Staubli VAL3: kernel.pjx

--- kernel.pjx ---
Parameters version=s7.7.2 stackSize=100000 millimeterUnit=true
Program file=_control.pgx
Program file=_cycle.pgx
Program file=_interface.pgx
Program file=_interfacePoint.pgx
Program file=_kill.pgx
Program file=_plc.pgx
Program file=_pointStep.pgx
Program file=_remote.pgx
Program file=_startCycle.pgx
Program file=_startSimul.pgx
Program file=_stopCycle.pgx
Program file=_stopSimul.pgx
Program file=_taskControl.pgx
Program file=action_buffer.pgx
Program file=action_bufferT.pgx
Program file=action_do.pgx
Program file=action_resume.pgx
Program file=action_suspend.pgx
Program file=action_wait.pgx
Program file=cycle_autoON.pgx
Program file=cycle_doEvent.pgx
Program file=cycle_init.pgx
Program file=cycle_isCallUse.pgx
Program file=cycle_run.pgx
Program file=cycle_simul.pgx
Program file=cycle_start.pgx
Program file=cycle_version.pgx
Program file=cycle_waitEmpty.pgx
Program file=memory_instr.pgx
Program file=memory_loadPage.pgx
Program file=memory_onEnd.pgx
Program file=memory_onRun.pgx
Program file=memory_onStop.pgx
Program file=memory_path.pgx
Program file=memory_reLoad.pgx
Program file=memory_showAll.pgx
Program file=memory_startUp.pgx
Program file=outOfRange.pgx
Program file=remote_isHome.pgx
Program file=remote_it.pgx
Program file=remote_loadHome.pgx
Program file=remote_rstLight.pgx
Program file=start.pgx
Program file=stop.pgx
Data file=kernel.dtx
Library alias=OnEvent path=Disk://OnEvent/OnEvent.pjx autoload=true password=
Library alias=saveData path=Disk://saveData/saveData.pjx autoload=true password=
Library alias=language path=Disk://kernel/language/language.pjx autoload=true password=
Library alias=use path=Disk://kernel/userPage/userPage.pjx autoload=true password=
Library alias=plc path=Disk://PLC/PLC.pjx autoload=true password=
Library alias=cycleStatus path=Disk://cycleStatus/cycleStatus.pjx autoload=true password=
Library alias=processList path=Disk://kernel/processList/processList.pjx autoload=true password=
Library alias=interface path=Disk://kernel/template/page/page.pjx autoload=true password=
Library alias=point_interface path=Disk://trajectory/page_trajectory/page_trajectory.pjx autoload=true password=
Library alias=inOut path=Disk://saveInputOutput/saveInputOutput.pjx autoload=true password=
Library alias=prog path=Disk://instruction/PROG/PROG.pjx autoload=true password=
Library alias=page0 path=./template/page/page.pjx autoload=true password=
Library alias=page1 path=./template/page/page.pjx autoload=true password=
Library alias=page2 path=./template/page/page.pjx autoload=true password=
Library alias=page3 path=./template/page/page.pjx autoload=true password=
Library alias=page4 path=./template/page/page.pjx autoload=true password=
Library alias=page5 path=./template/page/page.pjx autoload=true password=
Library alias=page6 path=./template/page/page.pjx autoload=true password=
Library alias=page7 path=./template/page/page.pjx autoload=true password=
Library alias=page8 path=./template/page/page.pjx autoload=true password=
Library alias=page9 path=./template/page/page.pjx autoload=true password=
Library alias=page10 path=./template/page/page.pjx autoload=true password=
Library alias=page11 path=./template/page/page.pjx autoload=true password=
Library alias=page12 path=./template/page/page.pjx autoload=true password=
Library alias=page13 path=./template/page/page.pjx autoload=true password=
Library alias=page14 path=./template/page/page.pjx autoload=true password=
Library alias=page15 path=./template/page/page.pjx autoload=true password=
Library alias=page16 path=./template/page/page.pjx autoload=true password=
Library alias=page17 path=./template/page/page.pjx autoload=true password=
Library alias=page18 path=./template/page/page.pjx autoload=true password=
Library alias=page19 path=./template/page/page.pjx autoload=true password=
Library alias=page20 path=./template/page/page.pjx autoload=true password=
Library alias=page21 path=./template/page/page.pjx autoload=true password=
Library alias=page22 path=./template/page/page.pjx autoload=true password=
Library alias=page23 path=./template/page/page.pjx autoload=true password=
Library alias=page24 path=./template/page/page.pjx autoload=true password=
Library alias=page25 path=./template/page/page.pjx autoload=true password=
Library alias=instr0 path=Disk://../templates/instruction/instruction.pjx autoload=true password=
Library alias=instr19 path=Disk://../templates/instruction/instruction.pjx autoload=true password=
Library alias=instr1 path=Disk://../templates/instruction/instruction.pjx autoload=true password=
Library alias=instr2 path=Disk://../templates/instruction/instruction.pjx autoload=true password=
Library alias=instr3 path=Disk://../templates/instruction/instruction.pjx autoload=true password=
Library alias=instr4 path=Disk://../templates/instruction/instruction.pjx autoload=true password=
Library alias=instr5 path=Disk://../templates/instruction/instruction.pjx autoload=true password=
Library alias=instr6 path=Disk://../templates/instruction/instruction.pjx autoload=true password=
Library alias=instr7 path=Disk://../templates/instruction/instruction.pjx autoload=true password=
Library alias=instr8 path=Disk://../templates/instruction/instruction.pjx autoload=true password=
Library alias=instr9 path=Disk://../templates/instruction/instruction.pjx autoload=true password=
Library alias=instr10 path=Disk://../templates/instruction/instruction.pjx autoload=true password=
Library alias=instr11 path=Disk://../templates/instruction/instruction.pjx autoload=true password=
Library alias=instr12 path=Disk://../templates/instruction/instruction.pjx autoload=true password=
Library alias=instr13 path=Disk://../templates/instruction/instruction.pjx autoload=true password=
Library alias=instr14 path=Disk://../templates/instruction/instruction.pjx autoload=true password=
Library alias=instr15 path=Disk://../templates/instruction/instruction.pjx autoload=true password=
Library alias=instr16 path=Disk://../templates/instruction/instruction.pjx autoload=true password=
Library alias=instr17 path=Disk://../templates/instruction/instruction.pjx autoload=true password=
Library alias=instr18 path=Disk://../templates/instruction/instruction.pjx autoload=true password=
Library alias=page path=./template/page/page.pjx autoload=true password=
Library alias=jHome path=./template/session/saveTraj/HOME/HOME.pjx autoload=true password=
Library alias=instr20 path=Disk://../templates/instruction/instruction.pjx autoload=true password=
Library alias=instr21 path=Disk://../templates/instruction/instruction.pjx autoload=true password=
Library alias=instr22 path=Disk://../templates/instruction/instruction.pjx autoload=true password=
Library alias=instr23 path=Disk://../templates/instruction/instruction.pjx autoload=true password=
Library alias=instr24 path=Disk://../templates/instruction/instruction.pjx autoload=true password=
Library alias=instr25 path=Disk://../templates/instruction/instruction.pjx autoload=true password=
Library alias=instr26 path=Disk://../templates/instruction/instruction.pjx autoload=true password=
Library alias=instr27 path=Disk://../templates/instruction/instruction.pjx autoload=true password=
Library alias=instr28 path=Disk://../templates/instruction/instruction.pjx autoload=true password=
Library alias=instr29 path=Disk://../templates/instruction/instruction.pjx autoload=true password=
Library alias=saveInOut path=Disk://saveInputOutput/saveInputOutput.pjx autoload=true password=
Type name=ActionItem path=./template/ActionItem/ActionItem.pjx
Type name=Instruction path=./template/Instruction/Instruction.pjx
Type name=InstrItem path=Disk://kernel/template/InstrItem/InstrItem.pjx
Type name=progItem path=./template/progItem/progItem.pjx
Type name=Trajectory path=./template/Trajectory/Trajectory.pjx
Type name=dioItem path=./template/dioItem/dioItem.pjx
Type name=TrajJointItem path=./template/TrajJointItem/TrajJointItem.pjx
Type name=TrajHome path=./template/TrajHome/TrajHome.pjx

--- kernel.dtx ---
bool bEdge[5]
bool bEmergency
bool bErrorLoading
bool bHold
bool bPowered
bool bQuit
bool bRestartMove
bool bTaskPoint
bool bTimeOut
bool bWait
num nCycleStep = 4
num nLastWorkingM = 1
num nPLCClock = 7973.286
num nRemoteClock = 7973.286
num nRemoteID = -1
num nTimeOut = 10
progItem pProg
  [0]
    InstrItem iEvent
      [0]
        string sData
        string sType
    string sID
string language
string sInstr
string sItem = "JOINT @HOME"
string sMessage
string sName
string sPageLoad
string sPath
string sPathInstr
string sPathTemplate = "Disk://kernel/template/"
string sRemoteID
string sVersion[13]
  [0] = "VAL3 - s6.3.1"
  [1] = "Option testMode - demo"
  [2] = "Option valPlast - demo"
  [3] = "Configuration - D24265574A"
  [4] = "SerialNumber - ?"
  [5] = "Arm - tx90-S1-R4"
  [6] = "ArmSerialNumber - ?"
  [7] = "EP - s6.3"
  [8] = "SCA - s6.3"
  [9] = "PLC - s6.3"
  [10] = "Options - s6.3"
  [11] = "Relbo - s6.2"
  [12] = "Relbo - s5.3.2"

--- start.pgx ---
public program start()
  local num i
  local num l_nKey
  local string l_sMessage
begin
  // set the language
  call language:setLanguage(language:libPath()+"/"+saveData:language)
  // check if the robot is calibrated
  if isCalibrated()
    // FIRST BOOT
    if saveData:bInitAll
      call inOut:resetAll()
    endIf
    // INIT
    title("")
    setTextMode(0)
    userPage()
    cls()
    // SEARCH AND LOAD THE INSTRUCTION
    call language:message(l_sMessage,13)
    call use:strfill(l_sMessage,36,l_sMessage)
    call use:type(0,13,l_sMessage)
    do
      delay(0.5)
      call use:type(36+i,13,".")
      i=(i+1)
      l_nKey=getKey()
    until i==4 or l_nKey==255
    // clear the 13 line
    call use:clear(0,13)
    // look for the escape button
    if l_nKey==255 or saveData:bInitAll
      //  search for new instruction
      call language:message(l_sMessage,14)
      call use:type(2,1,l_sMessage)
      taskCreate "BuildInstr",100,memory_instr(true)
      saveData:bInitAll=false
    else
      // load in the memory the instruction
      call language:message(l_sMessage,15)
      call use:type(2,1,l_sMessage)
      taskCreate "BuildInstr",100,memory_instr(false)
    endIf
    // wait all instruction all well build
    do
      delay(0.5)
      call use:type(30+i,1,".    ")
      i=(i+1)%5
      if taskStatus("BuildInstr")>1
        taskKill("BuildInstr")
        bErrorLoading=true
        logMsg("[KERNEL] SUPERVISOR: error on loading Instruction")
        return
      endIf
    until taskStatus("BuildInstr")==-1
    // init all the variable use to comunicate with the SuperV
    cycleStatus:nToSuperV=-2
    cycleStatus:nInterfaceToSV=-2
    nRemoteID=-2
    plc:nToSuperV=-2
    // CYCLE INIT
    call cycleStatus:init()
    //
    // TASK
    //
    // CUSTOM TASK
    call OnEvent:OnStartup()
    // INTERFACE
    $jogPage(false)
    interface:libLoad("kernel/page/home")
    call use:type(1,6," Loading TASK Interface ")
    taskCreate "Interface",60,interface:main()
    wait(taskStatus("Interface")==1)
    // REMOTE
    call use:type(1,7," Loading TASK Remote ")
    taskCreate "Remote",20,remote_it()
    wait(taskStatus("Remote")==1)
    // PLC
    saveData:bPlc=true
    if saveData:bPlc==true
      call use:type(1,8," Loading TASK PLC ")
      taskCreate "Plc",50,plc:Main()
      wait(taskStatus("Plc")==1)
    endIf
    // START ALL
    cycleStatus:nToSuperV=-1
    cycleStatus:nInterfaceToSV=-1
    nRemoteID=-1
    plc:nToSuperV=-1
    //
    do
      /////////////////////////////////////////////////////
      // COMUNICATION between tha TASK
      /////////////////////////////////////////////////////
      // INTERFACE
      call _interface()
      // CYCLE
      call _cycle()
      // PLC
      if saveData:bPlc
        call _plc()
      endIf
      // REMOTE
      call _remote()
      //////////////////////
      // CONTROL
      //////////////////////
      // TASK PROBLEM
      call _taskControl()
      // CONTROL
      call _control()
      //////////////////////
      // OTHER
      //////////////////////
      // point step control
      call _pointStep()
      // CUSTOM control
      call OnEvent:control()
      // interface management
      call _interfacePoint()
      delay(0)
      //
    until bQuit
  else
    // ROBOT NOT CALIBRATED
    call language:message(l_sMessage,16)
    popUpMsg(l_sMessage)
    bErrorLoading=true
    return
  endIf
  // bye
  call _kill()
end

--- _control.pgx ---
program _control()
  local bool l_bCycle
  local bool l_bSimulation
  local num l_nID
  local num l_nResult
  local string l_sEmpty
  local string l_sMessage[2]
  local string l_sProg
begin
  //
  // load in advance to keep time
  //
  if !cycleStatus:bCycle and !cycleStatus:bSimulation and cycleStatus:bMutex==false and use:nPage>=20 and use:nPage<=29
    l_nID=0
    call processList:getCycle(l_sProg,l_nID,l_nID,0,1)
    if l_sProg!="" and !bErrorLoading
      // load the init one
      call processList:getCycle(l_sProg,l_nID,l_nID,0,0)
      if l_sProg==""
        call processList:getCycle(l_sProg,l_nID,l_nID,0,1)
      endIf
      // load it
      call prog:getProgItem(cycleStatus:pCycleProg,l_sProg)
      if cycleStatus:pCycleProg.sID==""
        // remove from the list
        bErrorLoading=true
      endIf
    elseIf l_sProg==""
      // reset the PROGRAM elements..
      resize(cycleStatus:pCycleProg.iEvent,1,1)
      cycleStatus:pCycleProg.iEvent.sType=""
      cycleStatus:pCycleProg.iEvent.sData=""
      cycleStatus:pCycleProg.sID=""
    endIf
  else
    bErrorLoading=false
  endIf
  //
  // look for the cycleStatus
  //
  if cycleStatus:bCycle
    // or cycleStatus:bSimulation
    //
    // if the working mode is not in the local or remote mode
    //
    if nLastWorkingM!=cycleStatus:nWorkingMode
      logMsg("[KERNEL] SUPERVISOR:Change working mode")
      call OnEvent:OnCycleEvent(6)
      nLastWorkingM=cycleStatus:nWorkingMode
    endIf
    // look if the power is on
    if isPowered()==false
      if bPowered
        // set the bit
        bPowered=false
        // save the last joint position if it wasn't stopped
        call cycleStatus:recordPowerDown()
        logMsg("[KERNEL] SUPERVISOR:Power off")
        call OnEvent:OnCycleEvent(7)
      endIf
    else
      bPowered=true
    endIf
    //
    // if the robot was moving and you release the hold key
    //
    if cycleStatus:nWorkingStatus==2 and cycleStatus:nPoint>0
      if !bHold
        logMsg("[KERNEL] SUPERVISOR:Release move Hold")
        call OnEvent:OnCycleEvent(0)
        bHold=true
      endIf
    else
      if cycleStatus:nWorkingStatus!=2
        bHold=false
      endIf
    endIf
    //
    // check the emergency
    //
    if esStatus()==2
      if !bEmergency
        bEmergency=true
        // look if the emergency is active
        call language:message(l_sMessage,222)
        popUpMsg(l_sMessage)
        call OnEvent:OnCycleEvent(1)
        logMsg("[KERNEL] SUPERVISOR:Emergence press")
        if saveData:bStopToPowerOff
          if cycleStatus:bCycle
            // CYCLE
            call _stopCycle()
          elseIf cycleStatus:bSimulation
            // SIMULATION
            call _stopSimul()
          endIf
          return
        endIf
      endIf
    else
      bEmergency=false
    endIf
  else
    // RESET ALL THE BIT
    bPowered=false
    bEmergency=false
    bHold=false
    nLastWorkingM=cycleStatus:nWorkingMode
    // check if already home -> reset the jPowerDown
    if cycleStatus:bIsHome
      call cycleStatus:recordPowerDown()
    endIf
  endIf
  //
  // check the restart move procedure
  //
  if !cycleStatus:bWait and !cycleStatus:bPause and !cycleStatus:bPausePLC and !cycleStatus:bStop and cycleStatus:bMoveStopped
    // restart the move
    restartMove()
    if saveData:bDebug
      ? "MOTION Restart,"+toString(".3",clock()-cycleStatus:nTime)
    endIf
    cycleStatus:bMoveStopped=false
    cycleStatus:bMotionToken=false
  else
    // stop the move
    if (cycleStatus:bWait or cycleStatus:bPause or cycleStatus:bPausePLC or cycleStatus:bStop) and !cycleStatus:bMoveStopped
      if saveData:bDebug
        ? "MOTION stopped,"+toString(".3",clock()-cycleStatus:nTime)
      endIf
      cycleStatus:bMoveStopped=true
    endIf
  endIf
  //
  // time control
  //
  // check for the resume of the task
  if bTimeOut and !cycleStatus:bPause and !cycleStatus:bPausePLC
    // resume the task
    call action_resume()
  endIf
  // is waiting
  if (cycleStatus:bWait and !cycleStatus:bPause and !cycleStatus:bPausePLC)
    if !bWait
      bTimeOut=false
      bWait=true
      nTimeOut=clock()
    endIf
    // check the time and pause the cycle
    if (clock()-nTimeOut)>saveData:nTimeOut and !bTimeOut and saveData:nTimeOut>0
      bTimeOut=true
      // suspend all the task action
      call action_suspend()
      call OnEvent:OnCycleEvent(22)
    endIf
  else
    // reset the time
    bWait=false
  endIf
  //
  // STATUS CONTROL
  //
  // save the status and the working mode of the task in global
  //
  cycleStatus:nWorkingMode=workingMode(cycleStatus:nWorkingStatus)
  cycleStatus:nEmergency=esStatus()
  // CYCLE STATUS
  l_bCycle=taskStatus("Cycle")==1 or taskStatus("Cycle")==0
  // SIMULATION STATUS
  l_bSimulation=taskStatus("Simulation")==1 or taskStatus("Simulation")==0
  //
  // REFRESH and CYCLE status
  //
  if cycleStatus:bSimulation!=l_bSimulation
    // simulation
    cycleStatus:bSimulation=l_bSimulation
    // INIT ALL
    if !l_bSimulation
      // init all
      call cycle_init()
      l_sEmpty=""
      call memory_onStop(l_sEmpty)
    endIf
    use:bUseRefresh=true
  endIf
  if cycleStatus:bCycle!=l_bCycle
    // cycle
    cycleStatus:bCycle=l_bCycle
    if !l_bCycle
      // init all
      call cycle_init()
      l_sEmpty=""
      call memory_onStop(l_sEmpty)
      // check if reload the last process List saved
      if saveData:bReloadList
        call processList:loadProcessList(l_nResult)
        if l_nResult!=0
          // message
          call language:message(l_sMessage,-7)
          call language:message(l_sMessage[1],70)
          popUpMsg(l_sMessage+" "+l_sMessage[1])
        endIf
      endIf
    endIf
    use:bUseRefresh=true
  endIf
  // check if is need to reload ALL
  if saveData:bToReload and !cycleStatus:bCycle and !cycleStatus:bSimulation
    call memory_reLoad()
    saveData:bToReload=false
  endIf
end

--- _cycle.pgx ---
program _cycle()
  local bool bActive
  local bool l_bContinue
  local bool l_bTollerance
  local string l_sMessage
begin
  bActive=false
  //
  // STOP CYCLE
  //
  if cycleStatus:bToStop
    stopMove()
    if cycleStatus:bCycle
      call _stopCycle()
    else
      // SIMULATION
      if cycleStatus:bSimulation
        call _stopSimul()
      endIf
    endIf
    //  RESET
    cycleStatus:bToStop=false
    cycleStatus:nToSuperV=-1
    //
    // HOMING
    //
  elseIf cycleStatus:bToHome
    cycleStatus:bToHome=false
    if watch(cycleStatus:bSimulation==false and cycleStatus:bCycle==false,3)
      cycleStatus:sTraj=""
      cycleStatus:iToSuperV.sType="HOME"
      cycleStatus:iToSuperV.sData="simul"
      call _startSimul(cycleStatus:iToSuperV)
    endIf
    //
    // END CYCLE
    //
  elseIf cycleStatus:bToEnd==true
    cycleStatus:bToEnd=false
    // end the cycle
    if cycleStatus:bCycle and !cycleStatus:bEnding and esStatus()!=2
      logMsg("[KERNEL] CYCLE:Ending Cycle")
      cycleStatus:bEnding=true
      call OnEvent:OnCycleEvent(4)
    endIf
    //
    // START CYCLE
    //
  elseIf cycleStatus:bToStart==true
    cycleStatus:bToStart=false
    if taskStatus("Cycle")==-1
      call _startCycle()
      logMsg("[KERNEL] SUPERVISOR:Cycle>Start cycle")
    endIf
    //
    // PAUSE / RESUME
    //
  elseIf cycleStatus:bToPause
    cycleStatus:bToPause=false
    // PAUSE
    if !cycleStatus:bPause
      // pause the robot
      cycleStatus:bPause=true
      // stop the motion
      stopMove()
      if isPowered()
        call cycleStatus:recordPowerDown()
      endIf
      logMsg("[KERNEL] CYCLE:Pause the cycle")
      // onEvent
      call OnEvent:OnCycleEvent(2)
      // resume the cycle after a pause
    elseIf cycleStatus:bPause==true and cycleStatus:bMoveStopped==true and esStatus()!=2
      // check the tollerance if not do nothing
      call cycleStatus:checkTollerance(l_bTollerance)
      if (!isPowered() and !l_bTollerance and (cycleStatus:nWorkingMode==4 or cycleStatus:nWorkingMode==3))
        logMsg("[KERNEL] CYCLE:Error on Tollerance check during RESTART")
      else
        logMsg("[KERNEL] CYCLE:Restart the cycle")
        // on Event
        call OnEvent:OnCycleEvent(3)
        // restart, reset the bit for the pause
        cycleStatus:bPause=false
      endIf
    endIf
  else
    // check the auto_ON
    if cycleStatus:bAutoON
      cycleStatus:bAutoON=false
      call cycle_autoON(l_bContinue)
    endIf
    // SWITCH
    switch cycleStatus:nToSuperV
      case 0
        //
      break
      case 1
        //
      break
      case 2
        //
      break
      case 3
        //
      break
      case 4
        // OUT OF TIME
        call language:message(l_sMessage,230)
        popUpMsg(l_sMessage)
        if cycleStatus:bCycle
          //STOP CYCLE
          call _stopCycle()
        else
          if cycleStatus:bSimulation
            // STOP SIMULATION
            call _stopSimul()
          endIf
        endIf
        bActive=true
      break
      case 6
        // PAUSE CYCLE
        call OnEvent:pauseCycle()
        bActive=true
      break
      case 7
        // RESUME CYCLE
        call OnEvent:resumeCycle()
        bActive=true
      break
      default
      break
    endSwitch
  endIf
  // release
  if bActive
    cycleStatus:nToSuperV=-1
  endIf
  //
end

--- _interface.pgx ---
program _interface()
  local bool bActive
  local bool bStop
  local num i
  local string message
  local string sString
begin
  bActive=false
  switch cycleStatus:nInterfaceToSV
    case 0
      //
      // go to the production page
      //
      logMsg("[KERNEL] SUPERVISOR:Interface>Call Production page")
      bActive=true
    break
    case 1
      //
      //  Exit from KERNEL
      //
      bQuit=true
      bActive=true
    break
    case 2
      //
      //  Simulation of a program
      //
      call _startSimul(cycleStatus:iToSuperV)
      bActive=true
    break
    case 3
      //
      //  Simulation of an Event
      //
      call _startSimul(cycleStatus:iToSuperV)
      bActive=true
    break
    case 4
      //
      //  Timer simulation
      //
      cycleStatus:iToSuperV.sType="TIMER"
      cycleStatus:iToSuperV.sData="executing"
      call _startSimul(cycleStatus:iToSuperV)
      bActive=true
    break
    //
    // PLC
    //
    case 10
      // PLC activation
      logMsg("[KERNEL] SUPERVISOR:Interface>Start the Task PLC")
      plc:nToSuperV=-2
      taskCreate "Plc",50,plc:Main()
      saveData:bPlc=true
      plc:nToSuperV=-1
      bActive=true
    break
    case 11
      // PLC de-activation
      logMsg("[KERNEL] SUPERVISOR:Interface>Kill the Task PLC")
      taskKill("Plc")
      call plc:kill()
      saveData:bPlc=false
      bActive=true
    break
    default
      //
    break
  endSwitch
  // reset
  if bActive
    cycleStatus:nInterfaceToSV=-1
  endIf
end

--- _interfacePoint.pgx ---
program _interfacePoint()
  local string l_sMessage
begin
  //
  // acces to the point interface
  //
  if isKeyPressed(289) and (taskStatus("Point")==-1 or taskStatus("Point")>1)
    if (use:nPage>=100000 and use:nPage<=100009) or (use:nPage>=10000 and use:nPage<=10009)
      // TODO
      l_sMessage="Please exit from the page editor before enter in page POINT...."
      popUpMsg(l_sMessage)
      delay(3)
    else
      // SUSPEND THE TASK INTERFACE
      taskKill("Point")
      taskSuspend("Interface")
      // POINT INTERFACE
      taskCreate "Point",50,point_interface:main()
      bTaskPoint=true
      use:bUseRefresh=true
    endIf
  elseIf (taskStatus("Interface")==0 and taskStatus("Point")==-1) and bTaskPoint
    // TASK RESUME
    bTaskPoint=false
    taskResume("Interface",0)
    use:bUseRefresh=true
  endIf
  // release
  delay(0)
end

--- _kill.pgx ---
public program _kill()
  local string l_sMessage
begin
  // KILL KERNEL
  $jogPage(true)
  title("")
  cls()
  call language:message(l_sMessage,17)
  call use:timerDialog(l_sMessage,0)
  logMsg("[KERNEL] SUPERVISOR:Interface>Quit KERNEL")
  taskKill("Interface")
  taskKill("Point")
  taskKill("Remote")
  taskKill("Cycle")
  taskKill("Plc")
  taskKill("Action")
  watch(taskStatus("Interface")==-1,1)
  watch(taskStatus("Remote")==-1,1)
  watch(taskStatus("Cycle")==-1,1)
  watch(taskStatus("Plc")==-1,1)
  // save the last setting
  saveData:libSave()
  // save the cycle
  call processList:save()
  bQuit=false
  // give a time delay
  delay(1)
end

--- _plc.pgx ---
program _plc()
  local bool bActive
begin
  // PLC
  bActive=false
  switch plc:nToSuperV
    case 0
      //
      // Start Cycle
      //
      if taskStatus("Cycle")==-1
        cycleStatus:bToStart=true
      endIf
      bActive=true
    break
  endSwitch
  //
  if bActive
    plc:nToSuperV=-1
  endIf
end

--- _pointStep.pgx ---
program _pointStep()
  local ActionItem l_aPointData
  local num l_nId
  local num l_nIdPoint
  local num l_nLastId
  local Trajectory l_tTraj
begin
  //
  //  SYNCRO the point STEP of the trajectory
  //
  //  only if on Cycle
  if (cycleStatus:bCycle or cycleStatus:bSimulation)
    // get the actual Point ID..
    call cycleStatus:getTraj(l_tTraj)
    if l_tTraj.sID!="null" and l_tTraj.sID!=""
      // check it..
      if cycleStatus:nPoint>size(l_tTraj.tSuper)-1
        // init all
        cycleStatus:nPoint=0
        call cycleStatus:removeTraj()
        //? "[POINTSTEP]: trajectory removed:"+l_tTraj.sID
      elseIf getMoveId()>l_tTraj.tSuper[cycleStatus:nPoint].nMoveId+1
        //? "[POINTSTEP]: trajectory update: "+l_tTraj.sID+toString("4",cycleStatus:nPoint)
        // put one MORE
        cycleStatus:nPoint=cycleStatus:nPoint+1
      endIf
      if !isEmpty()
        // set a traj is doing
        cycleStatus:bTraj=true
        if cycleStatus:nEvent!=l_tTraj[0].nId
          // update the EVENT ID
          cycleStatus:nEvent=l_tTraj[0].nId
          //? "[POINTSTEP]: trajectory event update: "+l_tTraj.sID+toString("4",cycleStatus:nEvent)
        endIf
        l_nId=roundDown(getMoveId())
        // refresh the percentage point distance
        cycleStatus:nIdPercentage=abs(getMoveId()-l_nId)*100
      endIf
    elseIf cycleStatus:nPoint!=0 or cycleStatus:bTraj
      // reset
      //? "[POINTSTEP]: reset the traj parameter"
      cycleStatus:bTraj=false
      cycleStatus:nPoint=0
    endIf
  else
    // reset the TRAJ
    cycleStatus:nPoint=0
    cycleStatus:bTraj=false
  endIf
  //
end

--- _remote.pgx ---
program _remote()
  local bool bActive
  local InstrItem l_iProg
  local string message
  local string sString
begin
  bActive=false
  switch nRemoteID
    case 0
      // START
      if taskStatus("Cycle")==-1
        logMsg("[KERNEL] SUPERVISOR:REMOTE>Start cycle")
        cycleStatus:bToStart=true
      endIf
      bActive=true
    break
    case 1
      //STOP
      cycleStatus:bToStop=true
      bActive=true
    break
    case 2
      //END CYCLE
      if taskStatus("Cycle")!=-1
        logMsg("[KERNEL] SUPERVISOR:REMOTE>End cycle")
        cycleStatus:bToEnd=true
      endIf
      bActive=true
    break
    case 3
      // HOME STRATEGY
      if taskStatus("Cycle")==-1
        logMsg("[KERNEL] SUPERVISOR:REMOTE>Home strategy")
        cycleStatus:bToHome=true
      endIf
      bActive=true
    break
    case 4
      // simulation of the program
      l_iProg.sType="PROG"
      l_iProg.sData=sRemoteID
      call _startSimul(l_iProg)
      logMsg("[KERNEL] SUPERVISOR:REMOTE>insert the program: "+sRemoteID)
      bActive=true
    break
  endSwitch
  if bActive
    nRemoteID=-1
    sRemoteID=""
    if taskStatus("Interface")==0
      taskResume("Interface",0)
    endIf
  endIf
end

--- _startCycle.pgx ---
program _startCycle()
  local bool l_bContinue
  local num l_nID
  local string l_sMessage
  local string l_sProcessList
begin
  // check home
  if cycleStatus:bIsHome or saveData:bNoUseHome
    // look if there are program into the process list
    if !cycleStatus:bCycle and !cycleStatus:bSimulation and esStatus()!=2
      call processList:getLoaded(l_sProcessList)
      if l_sProcessList!=""
        l_nID=0
        call processList:getCycle(l_sMessage,l_nID,l_nID,0,1)
        if l_sMessage!=""
          // Create the Cycle Task
          if taskStatus("Cycle")==-1
            // init all
            call cycleStatus:init()
            // onEvent
            cycleStatus:bCycle=true
            call OnEvent:OnCycleEvent(13)
            if cycleStatus:bToStop
              cycleStatus:bCycle=false
              return
            endIf
            // put the power ON on remote
            call cycle_autoON(l_bContinue)
            if l_bContinue
              taskCreate "Cycle",80,cycle_start()
              // start the action Task for the traj
              if taskStatus("Action")==-1
                taskCreate "Action",80,action_buffer()
              endIf
            else
              // error while starting
              cycleStatus:bCycle=false
              return
            endIf
          endIf
        else
          // ERROR no program into the process list
          call OnEvent:OnCycleEvent(9)
        endIf
      else
        // NO processList loaded
        call OnEvent:OnCycleEvent(9)
      endIf
    endIf
  else
    // the robot is not at home
    call language:message(l_sMessage,223)
    popUpMsg(l_sMessage)
  endIf
end

--- _startSimul.pgx ---
program _startSimul(InstrItem& x_iInstr (dimensions=1))
  local bool l_bContinue
  local string l_sEvent
begin
  // init all
  call cycleStatus:init()
  // CHECK FOR CYCLE EVENT
  if !cycleStatus:bCycle and !cycleStatus:bSimulation
    // set the Simulation is ON
    cycleStatus:bSimulation=true
    if x_iInstr.sType=="HOME"
      cycleStatus:bHoming=true
    endIf
    // SIMULATION
    logMsg("[KERNEL] SUPERVISOR:Interface>Simulation of the event: "+x_iInstr.sType+" "+x_iInstr.sData)
    taskCreate "Simulation",50,cycle_simul(x_iInstr)
    // start the action Task for the traj
    taskCreate "Action",80,action_buffer()
  endIf
end

--- _stopCycle.pgx ---
program _stopCycle()
  local string l_sEmpty
  local num nCycleDone
  local num nCycleToDo
  local string sProgName
begin
  // reset the bit
  // Stop the robot
  stopMove()
  if saveData:bStopToPowerOff
    disablePower()
  endIf
  logMsg("[KERNEL] SUPERVISOR:Cycle>Stop cycle")
  // kill the Task...
  taskKill("Cycle")
  taskKill("Action")
  watch(taskStatus("Cycle")==-1 and taskStatus("Action")==-1,1)
  //
  resetMotion()
  call OnEvent:OnCycleEvent(5)
  // delete the last program
  call processList:getCycle(sProgName,nCycleToDo,nCycleDone,0,1)
  if (nCycleToDo-nCycleDone)<=1
    call processList:loopMode()
  else
    call processList:setCycle(sProgName,nCycleToDo,nCycleDone+1,0,1)
  endIf
end

--- _stopSimul.pgx ---
program _stopSimul()
  local string l_sEmpty
begin
  // reset the bit
  stopMove()
  // STOP SIMULATION
  logMsg("[KERNEL] SUPERVISOR:Cycle>Stop Simulation")
  // kill the task...
  taskKill("Simulation")
  taskKill("Action")
  watch(taskStatus("Simulation")==-1 and taskStatus("Action")==-1,1)
  //
  resetMotion()
  call OnEvent:OnCycleEvent(10)
end

--- _taskControl.pgx ---
program _taskControl()
  local bool l_bRestart[2]
  local bool l_bYes
  local string l_sButton[2]
  local string l_sMessage[2]
begin
  //
  // Check the task Cycle
  //
  if taskStatus("Cycle")>1 or (cycleStatus:bCycle and taskStatus("Action")>1)
    if taskStatus("Cycle")>=150 and taskStatus("Cycle")<=154
      call outOfRange()
    else
      logMsg("[KERNEL] SUPERVISOR:Task Cycle problem")
      call OnEvent:OnCycleEvent(12)
    endIf
    call _stopCycle()
  endIf
  //
  // Check the task Simulation
  //
  if taskStatus("Simulation")>1 or (cycleStatus:bSimulation and taskStatus("Action")>1)
    if taskStatus("Simulation")>=150 and taskStatus("Simulation")<=154
      call outOfRange()
    else
      logMsg("[KERNEL] SUPERVISOR:Task Simulation problem")
      call OnEvent:OnCycleEvent(12)
    endIf
    call _stopSimul()
  endIf
  // Check the task PLC every 5 second
  if taskStatus("Plc")>1
    if clock()-nPLCClock>5
      nPLCClock=clock()
      taskResume("Plc",0)
    endIf
  else
    nPLCClock=clock()
  endIf
  // check the task remote every 5 seconds
  if taskStatus("Remote")>1
    if clock()-nRemoteClock>5
      nRemoteClock=clock()
      taskKill("Remote")
      taskCreate "Remote",20,remote_it()
    endIf
  else
    nRemoteClock=clock()
  endIf
  //
  // TASK INTERFACE
  //
  //
  // look if there is something wrong for the interface
  //
  l_bRestart=false
  if taskStatus("Interface")==61
    logMsg("[KERNEL] SUPERVISOR:WakeUpInterface> error61")
    get()
    taskResume("Interface",0)
    watch(taskStatus("Interface")==1,1)
  endIf
  //
  // look if the interface has been stopped
  //
  if cycleStatus:nInterfaceToSV==-1 and taskStatus("Simulation")==-1
    // look for the mode
    if taskStatus("Interface")>1
      call language:message(l_sMessage,221)
      call use:timerDialog(l_sMessage,1)
      // get a Key
      get()
      // RESTART ...
      logMsg("[KERNEL] SUPERVISOR:WakeUpInterface>Restart")
      call language:message(l_sMessage,220)
      call use:timerDialog(l_sMessage,1)
      taskKill("Interface")
      taskCreate "Interface",60,interface:main()
      wait(taskStatus("Interface")==1)
    endIf
  endIf
  //
  // look if the interface has been stopped
  //
  if cycleStatus:nInterfaceToSV==-1 and taskStatus("Simulation")==-1
    if taskStatus("Point")>1
      call language:message(l_sMessage,221)
      call use:timerDialog(l_sMessage,1)
      // get a Key
      get()
      // RESTART
      logMsg("[KERNEL] SUPERVISOR:WakeUpInterface>Restart Point")
      call language:message(l_sMessage,220)
      call use:timerDialog(l_sMessage,1)
      taskKill("Point")
      taskCreate "Point",50,point_interface:main()
      wait(taskStatus("Point")==1)
    endIf
  endIf
end

--- action_buffer.pgx ---
program action_buffer()
  local ActionItem l_aAction
  local bool l_bEmpty
begin
  // wait the Task Cycle or simulation has been started
  wait(cycleStatus:bCycle or cycleStatus:bSimulation)
  //
  // scan the action
  //
  while (cycleStatus:bCycle or cycleStatus:bSimulation)
    // wait to move to run STATE
    do
      // scan the action item
      call cycleStatus:isActionEmpty(l_bEmpty)
      cycleStatus:bActionRunning=!l_bEmpty
      if !(cycleStatus:bCycle or cycleStatus:bSimulation)
        return
      endIf
      delay(0)
    until l_bEmpty==false
    // execute
    call cycleStatus:getAction(l_aAction)
    call action_do(l_aAction,-1)
    // remove
    call cycleStatus:removeAction()
  endWhile
  //
end

--- action_bufferT.pgx ---
program action_bufferT(ActionItem& x_aAction[] (dimensions=1))
  local num i
  local bool l_bMutex
  local bool l_bTraj
  local num l_nActualStep
  local num l_nIdTask
  local num l_nInstrId
  local num l_nMinus
  local num l_nTask
  local num l_nZero
  local string l_sAction
  local string l_sEmpty
  local string l_sInstrType
begin
  //
  // INIT
  //
  // wait the Task Cycle or simulation has been started
  wait(cycleStatus:bCycle or cycleStatus:bSimulation)
  //
  if x_aAction.iInstr.sType!="" and x_aAction.iInstr.sType!="null"
    // compose the instruction
    // do the action
    x_aAction.nDistance=0
    x_aAction.nMoveId=-1
    x_aAction.nPointId=-1
    call action_do(x_aAction,-1)
  endIf
end

--- action_do.pgx ---
program action_do(ActionItem& x_aAction[] (dimensions=1), num x_nIndex (dimensions=1))
  local num i
  local num j
  local bool l_bExit
  local num l_nClock
  local num l_nDistance
  local num l_nResult
  local string l_sData
  local string l_sEmpty
  local string l_sInstr
  local string l_sInstruction
  local string l_sType
begin
  // check if not empty...
  if x_aAction.iInstr[0].sType!="" or x_aAction.iInstr[1].sType!="" or x_aAction.iInstr[2].sType!=""
    if saveData:bDebug
      ? "ACTION INSERT,"+x_aAction.iInstr.sType+" "+x_aAction.iInstr.sData+",ID="+toString(".3",getMoveId())+","+toString(".3",clock()-cycleStatus:nTime)+",x_ID="+toString("",x_aAction.nMoveId)+",x_Dist="+toString(".2",x_aAction.nDistance)
    endIf
    l_nClock=clock()
    // wait the correct moveID
    wait((x_aAction.nMoveId+x_aAction.nDistance)<=getMoveId() or (isEmpty()) and !cycleStatus:bPause)
    // look if there are several sAction in the traj
    for i=0 to (size(x_aAction.iInstr)-1)
      // check for not empty space
      if x_aAction.iInstr[i].sType!=""
        // get the instruction
        l_sData=x_aAction.iInstr[i].sData
        l_sType=x_aAction.iInstr[i].sType
        call saveInOut:replaceIO(l_sData,l_sType,l_sData)
        l_sInstr=l_sType+" "+l_sData
        if saveData:bDebug
          ? "ACTION RUNNING,"+l_sInstr+",ID="+toString(".3",getMoveId())+","+toString(".3",clock()-cycleStatus:nTime)+",MoveID="+toString("",x_aAction.nMoveId)+",Dist="+toString(".2",x_aAction.nDistance)
        endIf
        // PRINT LOG
        if cycleStatus:bCycle
          if x_aAction.nPointId!=-1
            // is inside a trajectory
            call cycleStatus:printLog(" ."+l_sInstr)
          else
            // is outside a trajectory
            call cycleStatus:printLog("-"+l_sInstr)
          endIf
        endIf
        cycleStatus:sToShow=l_sInstr
        cycleStatus:sLastAction=l_sInstr
        if x_aAction.nPointId==-1
          // refresh the LINE of the program...
          cycleStatus:bTraj=false
          cycleStatus:nEvent=x_nIndex
        endIf
        //
        // RUN THE ACTION
        //
        call memory_onRun(x_aAction.iInstr[i])
      endIf
    endFor
    // release
    cycleStatus:sToShow=""
  endIf
end

--- action_resume.pgx ---
program action_resume()
begin
  //
  // suspend all the task action
  //
  // check first...
  if taskStatus("Cycle")!=-1
    taskResume("Cycle",0)
  endIf
  if taskStatus("Action")!=-1
    taskResume("Action",0)
  endIf
  //..
end

--- action_suspend.pgx ---
program action_suspend()
begin
  // suspend all the task action
  if taskStatus("Cycle")!=-1
    taskSuspend("Cycle")
  endIf
  if taskStatus("Action")!=-1
    taskSuspend("Action")
  endIf
  //..

end

--- action_wait.pgx ---
program action_wait()
  local bool l_bEmpty
begin
  // wait no action on the list
  while l_bEmpty==false
    call cycleStatus:isActionEmpty(l_bEmpty)
    delay(0)
  endWhile
end

--- cycle_autoON.pgx ---
program cycle_autoON(bool& x_bResult[] (dimensions=1))
  local num i
  local bool l_bTollerance
  local num l_nClock
  local string l_sMessage
begin
  //
  // look first if is in remote mode then
  // look if it is in mode automatic and the power is ON
  //
  x_bResult=false
  //
  //  CHECK FOR STATUS MODE
  //
  // look for the remote status NB check jPowerDown
  if workingMode()==4
    // check tollerance
    call cycleStatus:checkTollerance(l_bTollerance)
    if (!isPowered() and !l_bTollerance and cycleStatus:bPause)
      logMsg("[KERNEL] CYCLE:Error on Tollerance check during AUTO ON")
    elseIf isPowered()==false and esStatus()!=2 and cycleStatus:nWorkingMode!=2
      // enable auto connect move
      autoConnectMove(true)
      // VAL3 ?? unknow
      x_bResult=true
      // power it
      enablePower()
      delay(1)
      watch((isPowered()==true or esStatus()==2),3)
      if esStatus()==2
        return
      endIf
    endIf
  elseIf workingMode()!=3
    // put the robot in AUTO MODE
    call language:message(l_sMessage,200)
    // look fot the auto mode
    call use:timerDialog(l_sMessage,2)
  elseIf workingMode()==3 and !isPowered()
    // pu the power ON
    call language:message(l_sMessage,201)
    l_nClock=clock()
    do
      call use:timerDialog(l_sMessage,0.5)
    until (clock()-l_nClock)>5 or getKey()==255 or esStatus()==2
    if isPowered()==false
      return
    endIf
  endIf
  // it's ok give it back
  if esStatus()!=2 and ((workingMode()==3 or workingMode()==4) and isPowered())
    x_bResult=true
  endIf
  //
end

--- cycle_doEvent.pgx ---
program cycle_doEvent(InstrItem x_iInstr (dimensions=1), num x_nIndex (dimensions=1))
  local ActionItem l_aAction
  local bool l_bTraj
  local num l_nId
  local num l_nOffset
  local num l_nResult
  local string l_sInstruction
  local string l_sName
  local string l_sPath
begin
  //
  // DIVIDE INTO trajectory or NOT
  //
  call saveData:getPathInstr(x_iInstr.sType,l_sPath)
  if l_sPath!=""
    // DIVIDE INSTRUCTION FROM TRAJECTORY
    if find(l_sPath,"trajectory")==-1
      // EXECUTE THE ACTION
      call action_wait()
      // UPDATE THE ACTION TO DO...
      l_aAction.nDistance=1-saveData:nRound/100
      call cycleStatus:getLastId(l_aAction.nMoveId)
      l_aAction.iInstr=x_iInstr
      l_aAction.nPointId=-1
      call action_do(l_aAction,x_nIndex)
    else
      // TRAJ
      // print the action log
      l_sInstruction=x_iInstr.sType+" "+x_iInstr.sData
      if cycleStatus:bCycle
        // set the clock end
        call cycleStatus:printLog("-"+l_sInstruction)
      endIf
      // update the LINE ID
      cycleStatus:nLastIdPoint=x_nIndex
      // run it
      call memory_onRun(x_iInstr)
    endIf
  else
    // PATH NOT FOUND
    cycleStatus:bToStop=true
  endIf
end

--- cycle_init.pgx ---
program cycle_init()
// initialization of the cycle
  local num hours
  local num i
  local num index
  local num l_nSize
begin
  //
  // watch all the instructin has been launched
  //
  // init all the mutex
  cycleStatus:bMutex=false
  // reset
  if saveData:bDebug
    logMsg("[DEBUG] CYCLE: INIT Started")
    ? "CYCLE: INIT Started "
  endIf
  //
  // init all the cyclestatus variable
  //
  call cycleStatus:init()
  //
  // reset the cycle DONE
  //
  call processList:init()
  // check the version status
  call cycle_version()
  if saveData:bDebug
    logMsg("[DEBUG] CYCLE: INIT Terminated")
    ? "CYCLE: INIT Terminated"
  endIf
  // reset all the internal BIT
  bWait=false
  bTimeOut=false
end

--- cycle_isCallUse.pgx ---
program cycle_isCallUse()
  local num l_nResult
  local progItem l_pProg
begin
  // JUMP CALL USED
  if cycleStatus:bCALL
    do
      // reset the BIT
      cycleStatus:bCALL=false
      if cycleStatus:iToSuperV.sType=="PROG"
        // load the SUB PROG
        call prog:getProgItem(pProg,cycleStatus:iToSuperV.sData)
        // check it
        if pProg.sID!=""
          call cycle_run(pProg)
        else
          // STOP ALL
          cycleStatus:bToStop=true
        endIf
        // came back and restore
      else
        // just the LINE
        call cycle_doEvent(cycleStatus:iToSuperV,0)
      endIf
      // NESTED....
    until cycleStatus:bCALL==false
  endIf
end

--- cycle_run.pgx ---
program cycle_run(progItem& x_pProgram[] (dimensions=1))
  local num i
  local num j
  local num l_nClock
  local num l_nResult
  local num l_nSize
  local progItem l_pProg
  local string l_sEvent
begin
  //
  // START
  //
  cycleStatus:nEvent=0
  cycleStatus:nPoint=0
  // refresh
  cycleStatus:pCycleProg=l_pProg=x_pProgram
  // check the cycle
  if cycleStatus:bCycle
    // print the actual program
    call cycleStatus:printLog("[PROG "+l_pProg.sID+"]")
  endIf
  l_nSize=size(l_pProg.iEvent)
  for i=0 to l_nSize-1
    // wait pause false before doing the next instruction
    wait(cycleStatus:bPause==false and isPowered() and cycleStatus:nWorkingStatus==0)
    if l_pProg.iEvent[i].sType!=""
      l_sEvent=l_pProg.iEvent[i].sType+" "+l_pProg.iEvent[i].sData
      if saveData:bDebug
        ? "ACTION READ,"+l_sEvent+",ID="+toString(".3",getMoveId())+","+toString(".3",clock()-cycleStatus:nTime)
      endIf
      call cycle_doEvent(l_pProg.iEvent[i],i)
      // JUMP CALL USED
      call cycle_isCallUse()
      // GOTO USED
      if cycleStatus:bGOTO
        // terminate this and run the GOTO
        i=l_nSize-1
      endIf
    endIf
  endFor
  // GOTO ...
  if cycleStatus:bGOTO
    // INIT
    cycleStatus:bGOTO=false
    call action_wait()
    if cycleStatus:iToSuperV.sType=="PROG"
      // run the GOTO FOR PROG
      call prog:getProgItem(l_pProg,cycleStatus:iToSuperV.sData)
      //use:bUseRefresh=true
      call cycle_run(l_pProg)
    else
      call cycle_doEvent(cycleStatus:iToSuperV,0)
      // JUMP CALL USED
      call cycle_isCallUse()
    endIf
  endIf
end

--- cycle_simul.pgx ---
program cycle_simul(InstrItem x_iEvent (dimensions=1))
  local bool l_bContinue
  local num l_nKey
  local num l_nLoading
  local num l_nResult
  local progItem l_pProg
  local string l_sItem
  local string l_sMessage
begin
  // reset the recording
  resetMotion()
  // set the program
  l_sItem=x_iEvent.sType+" "+x_iEvent.sData
  // check if the timer simulation has to be done
  if cycleStatus:nWorkingMode!=1
    // check the workingMode
    call cycle_autoON(l_bContinue)
  else
    l_bContinue=true
  endIf
  // init the time..
  cycleStatus:nTime=clock()
  if l_bContinue
    // INIT
    call cycle_version()
    // check compatibility
    if cycleStatus:nToSuperV!=4
      // do the request
      if cycleStatus:bHoming
        // before HOME strategy
        // get the program
        call prog:getProgItem(l_pProg,"HOME1")
        // for simulation large screen
        use:bUseRefresh=true
        wait(cycleStatus:nWorkingStatus==0)
        logMsg("[KERNEL] SIMULATION:Execute the program: HOME1")
        // run it
        call cycle_run(l_pProg)
        // wait the end
        call cycle_waitEmpty()
        // onCycleEvent
        call OnEvent:OnCycleEvent(20)
      endIf
      // is a PROGRAM
      if x_iEvent.sType=="PROG"
        // for simulation large screen
        use:bUseRefresh=true
        wait(cycleStatus:nWorkingStatus==0)
        // cycleEvent Simulation Started
        call OnEvent:OnCycleEvent(17)
        logMsg("[KERNEL] SIMULATION:Execute the program: "+x_iEvent.sData)
        // load it
        call prog:loadCycle(x_iEvent.sData,l_nLoading)
        if l_nLoading!=0
          // program not found...
          popUpMsg("program not found")
          return
        endIf
        // run it
        call prog:getProgItem(pProg,x_iEvent.sData)
        // check if not empty
        if pProg.iEvent.sType!=""
          call cycle_run(pProg)
        endIf
      else
        // IS AN EVENT
        if x_iEvent.sType!=""
          l_pProg.sID="simul"
          l_pProg.iEvent=x_iEvent
          // refresh
          use:bUseRefresh=true
          wait(cycleStatus:nWorkingStatus==0)
          if !cycleStatus:bHoming
            // cycleEvent Simulation Started
            call OnEvent:OnCycleEvent(17)
          endIf
          // run it
          call cycle_run(l_pProg)
        endIf
      endIf
      // ENDING
      if cycleStatus:bHoming
        // get the program
        call prog:getProgItem(l_pProg,"HOME2")
        // for simulation large screen
        use:bUseRefresh=true
        wait(cycleStatus:nWorkingStatus==0)
        logMsg("[KERNEL] SIMULATION:Execute the program: HOME2")
        // run it
        call cycle_run(l_pProg)
        // wait the end
        call cycle_waitEmpty()
        // end of Home simulation
        call OnEvent:OnCycleEvent(21)
      else
        // wait the end
        call cycle_waitEmpty()
        if saveData:bDebug
          ? "End of Simulation: "+l_sItem
        endIf
        call OnEvent:OnCycleEvent(18)
      endIf
      // End of all
      call memory_onEnd()
    endIf
  endIf
end

--- cycle_start.pgx ---
program cycle_start()
  local num i
  local bool l_bContinue
  local bool l_bLoop
  local num l_nDone
  local num l_nLoading
  local num l_nSize
  local num l_nTotal
  local string l_sEmpty
  local string l_sItem
  local string l_sLoadProg
  local string l_sMessage
begin
  //
  // INIT AND REFRESH
  //
  // START THE CYCLE....
  resetMotion()
  logMsg("[KERNEL] CYCLE:Ready to Start")
  call cycle_version()
  // check compatibility
  if cycleStatus:nToSuperV!=4
    // send the ready to go
    //
    //  INIT CYCLE
    //
    // INIT the action log
    call cycleStatus:init_logAction()
    do
      // get the size
      call processList:getSize(l_nSize,cycleStatus:nProcessType)
      // check the size
      if cycleStatus:nProg<l_nSize or (saveData:bPlcEnable and cycleStatus:nProcessType==1)
        // wait a program...
        if (saveData:bPlcEnable and cycleStatus:nProcessType==1)
          do
            call processList:getSize(l_nSize,1)
            if isEmpty() and cycleStatus:bWait==false and isPowered() and cycleStatus:nWorkingStatus==0
              call language:message(l_sMessage,33)
              call language:message(l_sItem,-18)
              l_sMessage=l_sMessage+l_sItem
              call language:message(l_sItem,70)
              l_sMessage=l_sMessage+" "+l_sItem
              cycleStatus:sToShow=l_sMessage
            endIf
            delay(0)
          until cycleStatus:nProg<l_nSize or cycleStatus:bEnding
        endIf
        // look if the hold key was pressed
        wait(cycleStatus:nWorkingStatus==0)
        //
        // START ALL THE PROGRAM IN THE PROCESS LIST
        //
        call processList:getCycle(l_sLoadProg,l_nTotal,l_nDone,cycleStatus:nProg,cycleStatus:nProcessType)
        for i=l_nDone to (l_nTotal-1)
          // update the value
          call processList:getCycle(l_sLoadProg,l_nTotal,l_nDone,cycleStatus:nProg,cycleStatus:nProcessType)
          // load it
          call prog:loadCycle(l_sLoadProg,l_nLoading)
          if l_nLoading!=0
            // program not found...
            popUpMsg("program not found")
            return
          endIf
          call prog:getProgItem(pProg,l_sLoadProg)
          logMsg("[KERNEL] CYCLE:Execute the program: "+l_sLoadProg)
          // DO THE REFRESH
          cycleStatus:nTime=clock()
          // PROGRAM STARTED
          call OnEvent:OnCycleEvent(19)
          //
          // RUN IT
          //
          call cycle_run(pProg)
          // update all the data
          cycleStatus:nCycleTime=clock()-cycleStatus:nTime
          //increase the prog done value
          call processList:increase(cycleStatus:nProcessType)
          // check the end of Cycle
          if cycleStatus:bEnding and cycleStatus:nProcessType!=2 and l_nSize==1
            // endCycle
            i=l_nTotal
          endIf
          // WELL DONE
          call OnEvent:OnCycleEvent(14)
          call memory_onEnd()
          // reloop
        endFor
        // UPDATE
        call processList:getLoop(l_bLoop)
        call processList:getSize(l_nSize,1)
        if cycleStatus:bEnding and cycleStatus:nProcessType==1 and ((l_bLoop and cycleStatus:nProg>=max(l_nSize-1,0)) or !l_bLoop)
          // endCycle
          cycleStatus:nProcessType=2
          cycleStatus:nProg=0
          l_sLoadProg=""
        else
          // update the list
          if cycleStatus:nProcessType==1
            // remove from the list
            call processList:loopMode()
          else
            // go to next one
            cycleStatus:nProg=cycleStatus:nProg+1
          endIf
        endIf
      else
        // clear the list go to next
        l_sLoadProg=""
        cycleStatus:nProg=0
        cycleStatus:nProcessType=cycleStatus:nProcessType+1
      endIf
      delay(0)
    until cycleStatus:nProcessType>2
    //
    // wait the end of all
    //
    call cycle_waitEmpty()
    call OnEvent:OnCycleEvent(8)
  else
    // no power
    call language:message(l_sMessage,230)
    popUpMsg(l_sMessage)
  endIf
end

--- cycle_version.pgx ---
program cycle_version()
  local num i
  local num j
  local num l_hours
  local string l_sMessage
begin
  //
  // template Version status
  //
  if getVersion("valTending")!="enabled"
    //
    l_hours=roundDown(clock()/3600000)
    if l_hours>=2
      cycleStatus:nToSuperV=4
      call language:message(l_sMessage,230)
      popUpMsg(l_sMessage)
      cycleStatus:bToStop=true
    endIf
  endIf
end

--- cycle_waitEmpty.pgx ---
program cycle_waitEmpty()
begin
  // MOTION
  waitEndMove()
  wait(isEmpty())
  // task event
  call action_wait()
  // set the last time measure
  cycleStatus:nLastTimer=clock()-cycleStatus:nClockAction
end

--- memory_instr.pgx ---
program memory_instr(bool x_bSearch (dimensions=1))
  local num i
  local bool l_bDone
  local num l_nFind
  local num l_nSize
  local string l_sEmpty
  local string l_sItem
  local string l_sKey
  local string l_sPath
begin
  //
  // INIT
  //
  if x_bSearch
    //
    // this procedure build the list of instruction
    //
    l_sPath=""
    l_sEmpty=""
    call use:stringCopy(l_sEmpty,sInstr)
    call use:stringCopy(l_sEmpty,sPathInstr)
    call use:stringCopy(l_sEmpty,saveData:sInstr)
    call use:stringCopy(l_sEmpty,saveData:sInstrOnPoint)
    call use:stringCopy(l_sEmpty,saveData:sPageLoad)
    // delete all the instruction Type...
    l_sKey=first(saveData:iInstruction)
    // search it
    while l_sKey!=""
      // delete ALL
      delete(saveData:iInstruction[l_sKey])
      l_sKey=first(saveData:iInstruction)
    endWhile
    // rebuild
    call memory_path(l_sPath,sPathInstr)
    // copy the all path
    call use:stringCopy(sPathInstr,sInstr)
    call use:stringCopy(l_sEmpty,saveData:sPageLoad)
    //
    // delete the instruction that contain the field "_" as
    // use for page or other folder
    //
    for i=0 to (size(sInstr)-1)
      // look for all the page
      if find(sInstr[i],"page/")!=-1 or find(sInstr[i],"page_")!=-1
        if saveData:sPageLoad!=""
          insert(saveData:sPageLoad[size(saveData:sPageLoad)])
        endIf
        saveData:sPageLoad[size(saveData:sPageLoad)-1]=sInstr[i]
      endIf
      // delete the prefix of the path
      if find(sInstr[i],"instruction/")!=-1
        sInstr[i]=right(sInstr[i],len(sInstr[i])-len("instruction/"))
      else
        if find(sInstr[i],"trajectory/")!=-1
          sInstr[i]=right(sInstr[i],len(sInstr[i])-len("trajectory/"))
        else
          // delete
          if size(sInstr)>1
            delete(sInstr[i])
            delete(sPathInstr[i])
          endIf
          i=i-1
        endIf
      endIf
      if i>=0
        if find(sInstr[i],"_")!=-1 or find(sInstr[i],"language")!=-1 or find(sInstr[i],"program")!=-1
          delete(sInstr[i])
          delete(sPathInstr[i])
          i=i-1
        endIf
      endIf
    endFor
    // go just to the children
    for i=0 to (size(sInstr)-2)
      if find(sPathInstr[i+1],sPathInstr[i]+"/")!=-1
        l_bDone=false
        l_sPath=sPathInstr[i]
        delete(sInstr[i])
        delete(sPathInstr[i])
        do
          if find(sPathInstr[i],l_sPath)!=-1
            sInstr[i]=right(sPathInstr[i],len(sPathInstr[i])-len(l_sPath)-1)
            if i>=size(sPathInstr)-1
              l_bDone=true
            else
              if find(sPathInstr[i+1],sPathInstr[i])!=-1
                l_bDone=true
                i=i-1
              else
                i=i+1
              endIf
            endIf
          else
            l_bDone=true
            i=i-1
          endIf
        until l_bDone or i>=size(sInstr)
      endIf
    endFor
    //
    // BUILT the instr type as collection into saveData
    //
    // init saveData
    call use:stringCopy(sInstr,saveData:sInstr)
    call use:stringCopy(sInstr,saveData:sInstrOnPoint)
    call use:stringCopy(l_sEmpty,saveData:sTrajType)
    for i=0 to size(sInstr)-1
      l_sItem=sInstr[i]
      // insert all the item
      insert(saveData:iInstruction[l_sItem])
      saveData:iInstruction[l_sItem].sPath=sPathInstr[i]
      saveData:iInstruction[l_sItem].sID=sInstr[i]
      saveData:iInstruction[l_sItem].nIndex=i
      saveData:iInstruction[l_sItem].bIsTraj=false
      // check for traj
      if find(sPathInstr[i],"trajectory/")!=-1
        saveData:iInstruction[l_sItem].bIsTraj=true
        saveData:sInstrOnPoint[i]=""
        if saveData:sTrajType!=""
          append(saveData:sTrajType)
        endIf
        saveData:sTrajType[size(saveData:sTrajType)-1]=l_sItem
        // REMOVE the IF PROG from the point
      elseIf l_sItem=="IF" or l_sItem=="PROG"
        saveData:sInstrOnPoint[i]=""
      endIf
    endFor
    // save it
    saveData:libSave()
  endIf
  // start UP
  call memory_startUp(x_bSearch)
  // load all the page in the ram
  call memory_loadPage()
end

--- memory_loadPage.pgx ---
program memory_loadPage()
  local num i
  local num j
  local num k
  local num l_nResult
  local num l_nSize
  local string l_sChar[4]
  local string l_sMessage
begin
  // INIT INSTRUCTION
  call language:message(l_sMessage,20)
  call use:typeLen(2,1,l_sMessage,30)
  call use:clear(0,3)
  l_sChar[0]="|"
  l_sChar[1]="/"
  l_sChar[2]="-"
  l_sChar[3]="\"
  l_nSize=size(saveData:sPageLoad)
  k=0
  // TO BE COMPATIBLE...
  for i=0 to l_nSize-1
    // print to screen
    j=j%4
    call use:type(0,4,l_sChar[j])
    j=j+1
    call use:typeLen(2,4,saveData:sPageLoad[i],38)
    switch k
      case 0
        l_nResult=page0:libLoad(saveData:sPageLoad[i])
      break
      case 1
        l_nResult=page1:libLoad(saveData:sPageLoad[i])
      break
      case 2
        l_nResult=page2:libLoad(saveData:sPageLoad[i])
      break
      case 3
        l_nResult=page3:libLoad(saveData:sPageLoad[i])
      break
      case 4
        l_nResult=page4:libLoad(saveData:sPageLoad[i])
      break
      case 5
        l_nResult=page5:libLoad(saveData:sPageLoad[i])
      break
      case 6
        l_nResult=page6:libLoad(saveData:sPageLoad[i])
      break
      case 7
        l_nResult=page7:libLoad(saveData:sPageLoad[i])
      break
      case 8
        l_nResult=page8:libLoad(saveData:sPageLoad[i])
      break
      case 9
        l_nResult=page9:libLoad(saveData:sPageLoad[i])
      break
      case 10
        l_nResult=page10:libLoad(saveData:sPageLoad[i])
      break
      case 11
        l_nResult=page11:libLoad(saveData:sPageLoad[i])
      break
      case 12
        l_nResult=page12:libLoad(saveData:sPageLoad[i])
      break
      case 13
        l_nResult=page13:libLoad(saveData:sPageLoad[i])
      break
      case 14
        l_nResult=page14:libLoad(saveData:sPageLoad[i])
      break
      case 15
        l_nResult=page15:libLoad(saveData:sPageLoad[i])
      break
      case 16
        l_nResult=page16:libLoad(saveData:sPageLoad[i])
      break
      case 17
        l_nResult=page17:libLoad(saveData:sPageLoad[i])
      break
      case 18
        l_nResult=page18:libLoad(saveData:sPageLoad[i])
      break
      case 19
        l_nResult=page19:libLoad(saveData:sPageLoad[i])
      break
      case 20
        l_nResult=page20:libLoad(saveData:sPageLoad[i])
      break
      case 21
        l_nResult=page21:libLoad(saveData:sPageLoad[i])
      break
      case 22
        l_nResult=page22:libLoad(saveData:sPageLoad[i])
      break
      case 23
        l_nResult=page23:libLoad(saveData:sPageLoad[i])
      break
      case 24
        l_nResult=page24:libLoad(saveData:sPageLoad[i])
      break
      case 25
        l_nResult=page25:libLoad(saveData:sPageLoad[i])
      break
    endSwitch
    logMsg("[KERNEL] MEMORY:LOADED page "+saveData:sPageLoad[i]+toString("3",l_nResult))
    if l_nResult==0
      k=k+1
    endIf
    delay(0)
  endFor
  //
  call use:clear(0,4)
end

--- memory_onEnd.pgx ---
program memory_onEnd()
  local num i
  local num l_nSize
  local num l_nTime
  local string l_sEmpty
  local string l_sEvent
  local string l_sKey
begin
  //
  l_nTime=clock()
  //
  //
  l_sKey=first(saveData:iInstruction)
  // search it
  while l_sKey!="" and isDefined(saveData:iInstruction[l_sKey])
    switch saveData:iInstruction[l_sKey].nIndex
      case 0
        if instr0:libPath()!=""
          call instr0:onProgEnd(l_sEvent)
        endIf
      break
      case 1
        if instr1:libPath()!=""
          call instr1:onProgEnd(l_sEvent)
        endIf
      break
      case 2
        if instr2:libPath()!=""
          call instr2:onProgEnd(l_sEvent)
        endIf
      break
      case 3
        if instr3:libPath()!=""
          call instr3:onProgEnd(l_sEvent)
        endIf
      break
      case 4
        if instr4:libPath()!=""
          call instr4:onProgEnd(l_sEvent)
        endIf
      break
      case 5
        if instr5:libPath()!=""
          call instr5:onProgEnd(l_sEvent)
        endIf
      break
      case 6
        if instr6:libPath()!=""
          call instr6:onProgEnd(l_sEvent)
        endIf
      break
      case 7
        if instr7:libPath()!=""
          call instr7:onProgEnd(l_sEvent)
        endIf
      break
      case 8
        if instr8:libPath()!=""
          call instr8:onProgEnd(l_sEvent)
        endIf
      break
      case 9
        if instr9:libPath()!=""
          call instr9:onProgEnd(l_sEvent)
        endIf
      break
      case 10
        if instr10:libPath()!=""
          call instr10:onProgEnd(l_sEvent)
        endIf
      break
      case 11
        if instr11:libPath()!=""
          call instr11:onProgEnd(l_sEvent)
        endIf
      break
      case 12
        if instr12:libPath()!=""
          call instr12:onProgEnd(l_sEvent)
        endIf
      break
      case 13
        if instr13:libPath()!=""
          call instr13:onProgEnd(l_sEvent)
        endIf
      break
      case 14
        if instr14:libPath()!=""
          call instr14:onProgEnd(l_sEvent)
        endIf
      break
      case 15
        if instr15:libPath()!=""
          call instr15:onProgEnd(l_sEvent)
        endIf
      break
      case 16
        if instr16:libPath()!=""
          call instr16:onProgEnd(l_sEvent)
        endIf
      break
      case 17
        if instr17:libPath()!=""
          call instr17:onProgEnd(l_sEvent)
        endIf
      break
      case 18
        if instr18:libPath()!=""
          call instr18:onProgEnd(l_sEvent)
        endIf
      break
      case 19
        if instr19:libPath()!=""
          call instr19:onProgEnd(l_sEvent)
        endIf
      break
      case 20
        if instr20:libPath()!=""
          call instr20:onProgEnd(l_sEvent)
        endIf
      break
      case 21
        if instr21:libPath()!=""
          call instr21:onProgEnd(l_sEvent)
        endIf
      break
      case 22
        if instr22:libPath()!=""
          call instr22:onProgEnd(l_sEvent)
        endIf
      break
      case 23
        if instr23:libPath()!=""
          call instr23:onProgEnd(l_sEvent)
        endIf
      break
      case 24
        if instr24:libPath()!=""
          call instr24:onProgEnd(l_sEvent)
        endIf
      break
      case 25
        if instr25:libPath()!=""
          call instr25:onProgEnd(l_sEvent)
        endIf
      break
      case 26
        if instr26:libPath()!=""
          call instr26:onProgEnd(l_sEvent)
        endIf
      break
      case 27
        if instr27:libPath()!=""
          call instr27:onProgEnd(l_sEvent)
        endIf
      break
      case 28
        if instr28:libPath()!=""
          call instr28:onProgEnd(l_sEvent)
        endIf
      break
      case 29
        if instr29:libPath()!=""
          call instr29:onProgEnd(l_sEvent)
        endIf
      break
    endSwitch
    l_sKey=next(saveData:iInstruction[l_sKey])
  endWhile
  //
  if saveData:bDebug
    logMsg("[DEBUG] MEMORY:Charged all onProgEnd function using time: "+toString(".3",clock()-l_nTime))
  endIf
end

--- memory_onRun.pgx ---
program memory_onRun(InstrItem x_iInstr (dimensions=1))
  local Instruction l_iInstruction
  local num l_nResult
  local string l_sPath
begin
  //
  // load the instruction
  //
  if isDefined(saveData:iInstruction[x_iInstr.sType])
    switch saveData:iInstruction[x_iInstr.sType].nIndex
      case 0
        if instr0:libPath()!=""
          call instr0:onRun(x_iInstr.sData)
        endIf
      break
      case 1
        if instr1:libPath()!=""
          call instr1:onRun(x_iInstr.sData)
        endIf
      break
      case 2
        if instr2:libPath()!=""
          call instr2:onRun(x_iInstr.sData)
        endIf
      break
      case 3
        if instr3:libPath()!=""
          call instr3:onRun(x_iInstr.sData)
        endIf
      break
      case 4
        if instr4:libPath()!=""
          call instr4:onRun(x_iInstr.sData)
        endIf
      break
      case 5
        if instr5:libPath()!=""
          call instr5:onRun(x_iInstr.sData)
        endIf
      break
      case 6
        if instr6:libPath()!=""
          call instr6:onRun(x_iInstr.sData)
        endIf
      break
      case 7
        if instr7:libPath()!=""
          call instr7:onRun(x_iInstr.sData)
        endIf
      break
      case 8
        if instr8:libPath()!=""
          call instr8:onRun(x_iInstr.sData)
        endIf
      break
      case 9
        if instr9:libPath()!=""
          call instr9:onRun(x_iInstr.sData)
        endIf
      break
      case 10
        if instr10:libPath()!=""
          call instr10:onRun(x_iInstr.sData)
        endIf
      break
      case 11
        if instr11:libPath()!=""
          call instr11:onRun(x_iInstr.sData)
        endIf
      break
      case 12
        if instr12:libPath()!=""
          call instr12:onRun(x_iInstr.sData)
        endIf
      break
      case 13
        if instr13:libPath()!=""
          call instr13:onRun(x_iInstr.sData)
        endIf
      break
      case 14
        if instr14:libPath()!=""
          call instr14:onRun(x_iInstr.sData)
        endIf
      break
      case 15
        if instr15:libPath()!=""
          call instr15:onRun(x_iInstr.sData)
        endIf
      break
      case 16
        if instr16:libPath()!=""
          call instr16:onRun(x_iInstr.sData)
        endIf
      break
      case 17
        if instr17:libPath()!=""
          call instr17:onRun(x_iInstr.sData)
        endIf
      break
      case 18
        if instr18:libPath()!=""
          call instr18:onRun(x_iInstr.sData)
        endIf
      break
      case 19
        if instr19:libPath()!=""
          call instr19:onRun(x_iInstr.sData)
        endIf
      break
      case 20
        if instr20:libPath()!=""
          call instr20:onRun(x_iInstr.sData)
        endIf
      break
      case 21
        if instr21:libPath()!=""
          call instr21:onRun(x_iInstr.sData)
        endIf
      break
      case 22
        if instr22:libPath()!=""
          call instr22:onRun(x_iInstr.sData)
        endIf
      break
      case 23
        if instr23:libPath()!=""
          call instr23:onRun(x_iInstr.sData)
        endIf
      break
      case 24
        if instr24:libPath()!=""
          call instr24:onRun(x_iInstr.sData)
        endIf
      break
      case 25
        if instr25:libPath()!=""
          call instr25:onRun(x_iInstr.sData)
        endIf
      break
      case 26
        if instr26:libPath()!=""
          call instr26:onRun(x_iInstr.sData)
        endIf
      break
      case 27
        if instr27:libPath()!=""
          call instr27:onRun(x_iInstr.sData)
        endIf
      break
      case 28
        if instr28:libPath()!=""
          call instr28:onRun(x_iInstr.sData)
        endIf
      break
      case 29
        if instr29:libPath()!=""
          call instr29:onRun(x_iInstr.sData)
        endIf
      break
    endSwitch
  else
    // error instruction
    popUpMsg("INSTRUCTION NOT DEFINE !!!")
    cycleStatus:bToStop=true
  endIf
end

--- memory_onStop.pgx ---
program memory_onStop(string& x_sEvent[] (dimensions=1))
  local num i
  local num l_nSize
  local num l_nTime
  local string l_sKey
begin
  //
  // reload all the template...
  l_nTime=clock()
  //
  // find the instruction...
  l_sKey=first(saveData:iInstruction)
  // search it
  while l_sKey!="" and isDefined(saveData:iInstruction[l_sKey])
    switch saveData:iInstruction[l_sKey].nIndex
      case 0
        if instr0:libPath()!=""
          call instr0:onStop(x_sEvent)
        endIf
      break
      case 1
        if instr1:libPath()!=""
          call instr1:onStop(x_sEvent)
        endIf
      break
      case 2
        if instr2:libPath()!=""
          call instr2:onStop(x_sEvent)
        endIf
      break
      case 3
        if instr3:libPath()!=""
          call instr3:onStop(x_sEvent)
        endIf
      break
      case 4
        if instr4:libPath()!=""
          call instr4:onStop(x_sEvent)
        endIf
      break
      case 5
        if instr5:libPath()!=""
          call instr5:onStop(x_sEvent)
        endIf
      break
      case 6
        if instr6:libPath()!=""
          call instr6:onStop(x_sEvent)
        endIf
      break
      case 7
        if instr7:libPath()!=""
          call instr7:onStop(x_sEvent)
        endIf
      break
      case 8
        if instr8:libPath()!=""
          call instr8:onStop(x_sEvent)
        endIf
      break
      case 9
        if instr9:libPath()!=""
          call instr9:onStop(x_sEvent)
        endIf
      break
      case 10
        if instr10:libPath()!=""
          call instr10:onStop(x_sEvent)
        endIf
      break
      case 11
        if instr11:libPath()!=""
          call instr11:onStop(x_sEvent)
        endIf
      break
      case 12
        if instr12:libPath()!=""
          call instr12:onStop(x_sEvent)
        endIf
      break
      case 13
        if instr13:libPath()!=""
          call instr13:onStop(x_sEvent)
        endIf
      break
      case 14
        if instr14:libPath()!=""
          call instr14:onStop(x_sEvent)
        endIf
      break
      case 15
        if instr15:libPath()!=""
          call instr15:onStop(x_sEvent)
        endIf
      break
      case 16
        if instr16:libPath()!=""
          call instr16:onStop(x_sEvent)
        endIf
      break
      case 17
        if instr17:libPath()!=""
          call instr17:onStop(x_sEvent)
        endIf
      break
      case 18
        if instr18:libPath()!=""
          call instr18:onStop(x_sEvent)
        endIf
      break
      case 19
        if instr19:libPath()!=""
          call instr19:onStop(x_sEvent)
        endIf
      break
      case 20
        if instr20:libPath()!=""
          call instr20:onStop(x_sEvent)
        endIf
      break
      case 21
        if instr21:libPath()!=""
          call instr21:onStop(x_sEvent)
        endIf
      break
      case 22
        if instr22:libPath()!=""
          call instr22:onStop(x_sEvent)
        endIf
      break
      case 23
        if instr23:libPath()!=""
          call instr23:onStop(x_sEvent)
        endIf
      break
      case 24
        if instr24:libPath()!=""
          call instr24:onStop(x_sEvent)
        endIf
      break
      case 25
        if instr25:libPath()!=""
          call instr25:onStop(x_sEvent)
        endIf
      break
      case 26
        if instr26:libPath()!=""
          call instr26:onStop(x_sEvent)
        endIf
      break
      case 27
        if instr27:libPath()!=""
          call instr27:onStop(x_sEvent)
        endIf
      break
      case 28
        if instr28:libPath()!=""
          call instr28:onStop(x_sEvent)
        endIf
      break
      case 29
        if instr29:libPath()!=""
          call instr29:onStop(x_sEvent)
        endIf
      break
    endSwitch
    l_sKey=next(saveData:iInstruction[l_sKey])
    delay(0)
  endWhile
  if x_sEvent=="kill"
    // load the template for the session
    instr0:libLoad("Disk://../templates/instruction")
    delay(0)
    instr1:libLoad("Disk://../templates/instruction")
    delay(0)
    instr2:libLoad("Disk://../templates/instruction")
    delay(0)
    instr3:libLoad("Disk://../templates/instruction")
    delay(0)
    instr4:libLoad("Disk://../templates/instruction")
    delay(0)
    instr5:libLoad("Disk://../templates/instruction")
    delay(0)
    instr6:libLoad("Disk://../templates/instruction")
    delay(0)
    instr7:libLoad("Disk://../templates/instruction")
    delay(0)
    instr8:libLoad("Disk://../templates/instruction")
    delay(0)
    instr9:libLoad("Disk://../templates/instruction")
    delay(0)
    instr10:libLoad("Disk://../templates/instruction")
    delay(0)
    instr11:libLoad("Disk://../templates/instruction")
    delay(0)
    instr12:libLoad("Disk://../templates/instruction")
    delay(0)
    instr13:libLoad("Disk://../templates/instruction")
    delay(0)
    instr14:libLoad("Disk://../templates/instruction")
    delay(0)
    instr15:libLoad("Disk://../templates/instruction")
    delay(0)
    instr16:libLoad("Disk://../templates/instruction")
    delay(0)
    instr17:libLoad("Disk://../templates/instruction")
    delay(0)
    instr18:libLoad("Disk://../templates/instruction")
    delay(0)
    instr19:libLoad("Disk://../templates/instruction")
    delay(0)
    instr20:libLoad("Disk://../templates/instruction")
    delay(0)
    instr21:libLoad("Disk://../templates/instruction")
    delay(0)
    instr22:libLoad("Disk://../templates/instruction")
    delay(0)
    instr23:libLoad("Disk://../templates/instruction")
    delay(0)
    instr24:libLoad("Disk://../templates/instruction")
    delay(0)
    instr25:libLoad("Disk://../templates/instruction")
    delay(0)
    instr26:libLoad("Disk://../templates/instruction")
    delay(0)
    instr27:libLoad("Disk://../templates/instruction")
    delay(0)
    instr28:libLoad("Disk://../templates/instruction")
    delay(0)
    instr29:libLoad("Disk://../templates/instruction")
    delay(0)
  endIf
  //
  if saveData:bDebug
    logMsg("[DEBUG] MEMORY:Charged all onStop function using time: "+toString(".3",clock()-l_nTime))
  endIf
end

--- memory_path.pgx ---
program memory_path(string x_sPath (dimensions=1), string& x_sFolders[] (dimensions=1))
  local num i
  local num l_nSize
  local string l_sEmpty
  local string l_sPath
begin
  //
  // make o recursive all the path
  //
  l_sEmpty=""
  call use:stringCopy(l_sEmpty,sPath)
  libList(x_sPath,sPath)
  l_nSize=size(sPath)-1
  if sPath!=""
    for i=0 to l_nSize
      if find(sPath[i],".")==-1
        // compose
        l_sPath=x_sPath
        if x_sPath!=""
          // deepest
          x_sPath=x_sPath+"/"+sPath[i]
        else
          x_sPath=sPath[i]
        endIf
        //
        // increase the x_sFolders
        //
        if x_sFolders!=""
          insert(x_sFolders[size(x_sFolders)])
        endIf
        x_sFolders[size(x_sFolders)-1]=x_sPath
        //
        call memory_path(x_sPath,x_sFolders)
        // refresh the global variable
        l_sEmpty=""
        call use:stringCopy(l_sEmpty,sPath)
        libList(l_sPath,sPath)
        x_sPath=l_sPath
        //
      endIf
    endFor
  endIf
end

--- memory_reLoad.pgx ---
program memory_reLoad()
  local Instruction l_iInstruction
  local num l_nResult
  local string l_sKey
  local string l_sPath
begin
  //
  // load the instruction
  //
  //
  // find the instruction...
  l_sKey=first(saveData:iInstruction)
  // search it
  while l_sKey!="" and isDefined(saveData:iInstruction[l_sKey])
    l_nResult=0
    switch saveData:iInstruction[l_sKey].nIndex
      case 0
        if instr0:libPath()!=""
          call instr0:load("",l_nResult)
        endIf
      break
      case 1
        if instr1:libPath()!=""
          call instr1:load("",l_nResult)
        endIf
      break
      case 2
        if instr2:libPath()!=""
          call instr2:load("",l_nResult)
        endIf
      break
      case 3
        if instr3:libPath()!=""
          call instr3:load("",l_nResult)
        endIf
      break
      case 4
        if instr4:libPath()!=""
          call instr4:load("",l_nResult)
        endIf
      break
      case 5
        if instr5:libPath()!=""
          call instr5:load("",l_nResult)
        endIf
      break
      case 6
        if instr6:libPath()!=""
          call instr6:load("",l_nResult)
        endIf
      break
      case 7
        if instr7:libPath()!=""
          call instr7:load("",l_nResult)
        endIf
      break
      case 8
        if instr8:libPath()!=""
          call instr8:load("",l_nResult)
        endIf
      break
      case 9
        if instr9:libPath()!=""
          call instr9:load("",l_nResult)
        endIf
      break
      case 10
        if instr10:libPath()!=""
          call instr10:load("",l_nResult)
        endIf
      break
      case 11
        if instr11:libPath()!=""
          call instr11:load("",l_nResult)
        endIf
      break
      case 12
        if instr12:libPath()!=""
          call instr12:load("",l_nResult)
        endIf
      break
      case 13
        if instr13:libPath()!=""
          call instr13:load("",l_nResult)
        endIf
      break
      case 14
        if instr14:libPath()!=""
          call instr14:load("",l_nResult)
        endIf
      break
      case 15
        if instr15:libPath()!=""
          call instr15:load("",l_nResult)
        endIf
      break
      case 16
        if instr16:libPath()!=""
          call instr16:load("",l_nResult)
        endIf
      break
      case 17
        if instr17:libPath()!=""
          call instr17:load("",l_nResult)
        endIf
      break
      case 18
        if instr18:libPath()!=""
          call instr18:load("",l_nResult)
        endIf
      break
      case 19
        if instr19:libPath()!=""
          call instr19:load("",l_nResult)
        endIf
      break
      case 20
        if instr20:libPath()!=""
          call instr20:load("",l_nResult)
        endIf
      break
      case 21
        if instr21:libPath()!=""
          call instr21:load("",l_nResult)
        endIf
      break
      case 22
        if instr22:libPath()!=""
          call instr22:load("",l_nResult)
        endIf
      break
      case 23
        if instr23:libPath()!=""
          call instr23:load("",l_nResult)
        endIf
      break
      case 24
        if instr24:libPath()!=""
          call instr24:load("",l_nResult)
        endIf
      break
      case 25
        if instr25:libPath()!=""
          call instr25:load("",l_nResult)
        endIf
      break
      case 26
        if instr26:libPath()!=""
          call instr26:load("",l_nResult)
        endIf
      break
      case 27
        if instr27:libPath()!=""
          call instr27:load("",l_nResult)
        endIf
      break
      case 28
        if instr28:libPath()!=""
          call instr28:load("",l_nResult)
        endIf
      break
      case 29
        if instr29:libPath()!=""
          call instr29:load("",l_nResult)
        endIf
      break
    endSwitch
    // TODO
    if l_nResult!=0
      popUpMsg("instruction PROBLEM on reloading..."+l_sKey)
      logMsg("instruction PROBLEM on reloading..."+l_sKey)
    endIf
    // continue
    l_sKey=next(saveData:iInstruction[l_sKey])
  endWhile
end

--- memory_showAll.pgx ---
public program memory_showAll()
begin
  //
  // show all the path
  //
  logMsg("PAGE")
  logMsg(page0:libPath())
  logMsg(page1:libPath())
  logMsg(page2:libPath())
  logMsg(page3:libPath())
  logMsg(page4:libPath())
  logMsg(page5:libPath())
  logMsg(page6:libPath())
  logMsg(page7:libPath())
  logMsg(page8:libPath())
  logMsg(page9:libPath())
  logMsg(page10:libPath())
  logMsg(page11:libPath())
  logMsg(page12:libPath())
  logMsg(page13:libPath())
  logMsg(page14:libPath())
  logMsg(page15:libPath())
  logMsg(page16:libPath())
  logMsg(page17:libPath())
  logMsg(page18:libPath())
  logMsg(page19:libPath())
  logMsg(page20:libPath())
  logMsg(page21:libPath())
  logMsg(page22:libPath())
  logMsg(page23:libPath())
  logMsg(page24:libPath())
  logMsg(page25:libPath())
  logMsg("INSTRUCTION")
  logMsg(instr0:libPath())
  logMsg(instr1:libPath())
  logMsg(instr2:libPath())
  logMsg(instr3:libPath())
  logMsg(instr4:libPath())
  logMsg(instr5:libPath())
  logMsg(instr6:libPath())
  logMsg(instr7:libPath())
  logMsg(instr8:libPath())
  logMsg(instr9:libPath())
  logMsg(instr10:libPath())
  logMsg(instr11:libPath())
  logMsg(instr12:libPath())
  logMsg(instr13:libPath())
  logMsg(instr14:libPath())
  logMsg(instr15:libPath())
  logMsg(instr16:libPath())
  logMsg(instr17:libPath())
  logMsg(instr18:libPath())
  logMsg(instr19:libPath())
  logMsg(instr20:libPath())
  logMsg(instr21:libPath())
  logMsg(instr22:libPath())
  logMsg(instr23:libPath())
  logMsg(instr24:libPath())
  logMsg(instr25:libPath())
  logMsg(instr26:libPath())
  logMsg(instr27:libPath())
  logMsg(instr28:libPath())
  logMsg(instr29:libPath())
end

--- memory_startUp.pgx ---
program memory_startUp(bool x_bSearch (dimensions=1))
  local num i
  local num j
  local num l_nResult
  local num l_nSize
  local string l_sChar[4]
  local string l_sItem
  local string l_sKey
  local string l_sMessage
  local string l_sPath
  local num z
begin
  // INIT INSTRUCTION
  call language:message(l_sMessage,18)
  call use:type(2,3,l_sMessage)
  l_sChar[0]="|"
  l_sChar[1]="/"
  l_sChar[2]="-"
  l_sChar[3]="\"
  l_nSize=size(saveData:sInstr[i])
  // init all ?
  if x_bSearch
    l_sItem="init"
  endIf
  // TO BE COMPATIBLE...
  for i=(l_nSize-1) to 0 step -1
    // print to screen
    call use:strfill(saveData:sInstr[i],7,l_sMessage)
    call use:type(30,3,l_sChar[j]+" "+l_sMessage)
    j=(j+1)%4
    //get the path
    call saveData:getPathInstr(saveData:sInstr[i],l_sPath)
    if l_sPath==""
      l_nResult=0
    else
      switch i
        case 0
          l_nResult=instr0:libLoad(l_sPath)
          logMsg("[KERNEL] MEMORY:result of "+l_sPath+" = "+toString("",l_nResult))
          if l_nResult==0
            call instr0:onStart(l_sItem)
          endIf
        break
        case 1
          l_nResult=instr1:libLoad(l_sPath)
          logMsg("[KERNEL] MEMORY:result of "+l_sPath+" = "+toString("",l_nResult))
          if l_nResult==0
            call instr1:onStart(l_sItem)
          endIf
        break
        case 2
          l_nResult=instr2:libLoad(l_sPath)
          logMsg("[KERNEL] MEMORY:result of "+l_sPath+" = "+toString("",l_nResult))
          if l_nResult==0
            call instr2:onStart(l_sItem)
          endIf
        break
        case 3
          l_nResult=instr3:libLoad(l_sPath)
          logMsg("[KERNEL] MEMORY:result of "+l_sPath+" = "+toString("",l_nResult))
          if l_nResult==0
            call instr3:onStart(l_sItem)
          endIf
        break
        case 4
          l_nResult=instr4:libLoad(l_sPath)
          logMsg("[KERNEL] MEMORY:result of "+l_sPath+" = "+toString("",l_nResult))
          if l_nResult==0
            call instr4:onStart(l_sItem)
          endIf
        break
        case 5
          l_nResult=instr5:libLoad(l_sPath)
          logMsg("[KERNEL] MEMORY:result of "+l_sPath+" = "+toString("",l_nResult))
          if l_nResult==0
            call instr5:onStart(l_sItem)
          endIf
        break
        case 6
          l_nResult=instr6:libLoad(l_sPath)
          logMsg("[KERNEL] MEMORY:result of "+l_sPath+" = "+toString("",l_nResult))
          if l_nResult==0
            call instr6:onStart(l_sItem)
          endIf
        break
        case 7
          l_nResult=instr7:libLoad(l_sPath)
          logMsg("[KERNEL] MEMORY:result of "+l_sPath+" = "+toString("",l_nResult))
          if l_nResult==0
            call instr7:onStart(l_sItem)
          endIf
        break
        case 8
          l_nResult=instr8:libLoad(l_sPath)
          logMsg("[KERNEL] MEMORY:result of "+l_sPath+" = "+toString("",l_nResult))
          if l_nResult==0
            call instr8:onStart(l_sItem)
          endIf
        break
        case 9
          l_nResult=instr9:libLoad(l_sPath)
          logMsg("[KERNEL] MEMORY:result of "+l_sPath+" = "+toString("",l_nResult))
          if l_nResult==0
            call instr9:onStart(l_sItem)
          endIf
        break
        case 10
          l_nResult=instr10:libLoad(l_sPath)
          logMsg("[KERNEL] MEMORY:result of "+l_sPath+" = "+toString("",l_nResult))
          if l_nResult==0
            call instr10:onStart(l_sItem)
          endIf
        break
        case 11
          l_nResult=instr11:libLoad(l_sPath)
          logMsg("[KERNEL] MEMORY:result of "+l_sPath+" = "+toString("",l_nResult))
          if l_nResult==0
            call instr11:onStart(l_sItem)
          endIf
        break
        case 12
          l_nResult=instr12:libLoad(l_sPath)
          logMsg("[KERNEL] MEMORY:result of "+l_sPath+" = "+toString("",l_nResult))
          if l_nResult==0
            call instr12:onStart(l_sItem)
          endIf
        break
        case 13
          l_nResult=instr13:libLoad(l_sPath)
          logMsg("[KERNEL] MEMORY:result of "+l_sPath+" = "+toString("",l_nResult))
          if l_nResult==0
            call instr13:onStart(l_sItem)
          endIf
        break
        case 14
          l_nResult=instr14:libLoad(l_sPath)
          logMsg("[KERNEL] MEMORY:result of "+l_sPath+" = "+toString("",l_nResult))
          if l_nResult==0
            call instr14:onStart(l_sItem)
          endIf
        break
        case 15
          l_nResult=instr15:libLoad(l_sPath)
          logMsg("[KERNEL] MEMORY:result of "+l_sPath+" = "+toString("",l_nResult))
          if l_nResult==0
            call instr15:onStart(l_sItem)
          endIf
        break
        case 16
          l_nResult=instr16:libLoad(l_sPath)
          logMsg("[KERNEL] MEMORY:result of "+l_sPath+" = "+toString("",l_nResult))
          if l_nResult==0
            call instr16:onStart(l_sItem)
          endIf
        break
        case 17
          l_nResult=instr17:libLoad(l_sPath)
          logMsg("[KERNEL] MEMORY:result of "+l_sPath+" = "+toString("",l_nResult))
          if l_nResult==0
            call instr17:onStart(l_sItem)
          endIf
        break
        case 18
          l_nResult=instr18:libLoad(l_sPath)
          logMsg("[KERNEL] MEMORY:result of "+l_sPath+" = "+toString("",l_nResult))
          if l_nResult==0
            call instr18:onStart(l_sItem)
          endIf
        break
        case 19
          l_nResult=instr19:libLoad(l_sPath)
          logMsg("[KERNEL] MEMORY:result of "+l_sPath+" = "+toString("",l_nResult))
          if l_nResult==0
            call instr19:onStart(l_sItem)
          endIf
        break
        case 20
          l_nResult=instr20:libLoad(l_sPath)
          logMsg("[KERNEL] MEMORY:result of "+l_sPath+" = "+toString("",l_nResult))
          if l_nResult==0
            call instr20:onStart(l_sItem)
          endIf
        break
        case 21
          l_nResult=instr21:libLoad(l_sPath)
          logMsg("[KERNEL] MEMORY:result of "+l_sPath+" = "+toString("",l_nResult))
          if l_nResult==0
            call instr21:onStart(l_sItem)
          endIf
        break
        case 22
          l_nResult=instr22:libLoad(l_sPath)
          logMsg("[KERNEL] MEMORY:result of "+l_sPath+" = "+toString("",l_nResult))
          if l_nResult==0
            call instr22:onStart(l_sItem)
          endIf
        break
        case 23
          l_nResult=instr23:libLoad(l_sPath)
          logMsg("[KERNEL] MEMORY:result of "+l_sPath+" = "+toString("",l_nResult))
          if l_nResult==0
            call instr23:onStart(l_sItem)
          endIf
        break
        case 24
          l_nResult=instr24:libLoad(l_sPath)
          logMsg("[KERNEL] MEMORY:result of "+l_sPath+" = "+toString("",l_nResult))
          if l_nResult==0
            call instr24:onStart(l_sItem)
          endIf
        break
        case 25
          l_nResult=instr25:libLoad(l_sPath)
          logMsg("[KERNEL] MEMORY:result of "+l_sPath+" = "+toString("",l_nResult))
          if l_nResult==0
            call instr25:onStart(l_sItem)
          endIf
        break
        case 26
          l_nResult=instr26:libLoad(l_sPath)
          logMsg("[KERNEL] MEMORY:result of "+l_sPath+" = "+toString("",l_nResult))
          if l_nResult==0
            call instr26:onStart(l_sItem)
          endIf
        break
        case 27
          l_nResult=instr27:libLoad(l_sPath)
          logMsg("[KERNEL] MEMORY:result of "+l_sPath+" = "+toString("",l_nResult))
          if l_nResult==0
            call instr27:onStart(l_sItem)
          endIf
        break
        case 28
          l_nResult=instr28:libLoad(l_sPath)
          logMsg("[KERNEL] MEMORY:result of "+l_sPath+" = "+toString("",l_nResult))
          if l_nResult==0
            call instr28:onStart(l_sItem)
          endIf
        break
        case 29
          l_nResult=instr29:libLoad(l_sPath)
          logMsg("[KERNEL] MEMORY:result of "+l_sPath+" = "+toString("",l_nResult))
          if l_nResult==0
            call instr29:onStart(l_sItem)
          endIf
        break
        default
        break
      endSwitch
    endIf
    // check for the result not allow to continue
    if l_nResult!=0
      popUpMsg("ERROR on "+l_sPath+" = "+toString("",l_nResult)+chr(10)+" STOP CYCLE !!!")
      // make it crash
      instr0:libLoad(l_sPath)
      call instr0:onRun(l_sChar)
    endIf
    delay(0)
  endFor
end

--- outOfRange.pgx ---
program outOfRange()
  local num i
  local num l_nPoint
  local num l_nStackPoint
  local string l_sMessage
  local string l_sTraj
begin
  // find which trajectory and which point
  wait(isSettled())
  l_sTraj=cycleStatus:sTraj
  //
  l_nPoint=cycleStatus:nPoint
  // call the onEvent
  call OnEvent:OnCycleEvent(11)
  // out of range
  call language:message(l_sMessage,-5)
  l_sMessage=l_sMessage+" "+l_sTraj+" POINT: "+toString("4",l_nPoint)
  popUpMsg(l_sMessage)
  logMsg("[KERNEL] trajectory:POINT OUT OF RANGE, "+l_sTraj+" POINT: "+toString("4",l_nPoint))
  //
end

--- remote_isHome.pgx ---
program remote_isHome()
  local joint l_jHere
  local num l_nResult
  local num l_nSize
  local string l_sItem
begin
  // look if home was loaded
  if (!cycleStatus:bHomeLoaded or jHome:libPath()=="" or find(jHome:libPath(),"template")!=-1) and saveData:bToReload==false
    call remote_loadHome(l_nResult)
  endIf
  // ok home is in the ram
  l_sItem="home"
  l_nSize=size(jHome:tTraj[l_sItem].tData)-1
  if l_nResult==0 and jHome:tTraj[l_sItem].tData[l_nSize].jJoint!={0,0,0,0,0,0}
    // check if the the robot is nearby
    if abs(herej()-jHome:tTraj[l_sItem].tData[l_nSize].jJoint)<{1,1,1,2,2,2}
      // the robot is at home
      cycleStatus:bIsHome=true
    else
      cycleStatus:bIsHome=false
    endIf
  else
    cycleStatus:bIsHome=false
  endIf
  //
end

--- remote_it.pgx ---
program remote_it()
  local num i
  local bool l_bClock
  local bool l_bEnd
  local bool l_bTollerance
  local num l_nClock
  local string l_sKey
  local string l_sPath
  local string l_sProg
begin
  //
  // INIT
  //
  // HOME
  //
  cycleStatus:bHomeLoaded=cycleStatus:bIsHome=false
  saveData:bChangeIO=false
  //
  // the Start-stop-end_cycle
  //
  wait(nRemoteID==-1)
  l_nClock=clock()
  //
  logMsg("[KERNEL] REMOTE:LOAD")

